//{attribute 'qualified_only'}
//{attribute 'strict'}
TYPE enumFailReportSeverity :
(
	Warning 	:= 0,
	Error		:= 1,
	Critical	:= 2
	
);
END_TYPE

(* stored: Version 1.1.0.1, ProductVersion 3.1.4024.3
   DUT enumFailReportSeverity: Id {9afb4833-917e-0b9f-0fa8-362b43c685e9} *)
